{attribute 'qualified_only'}
VAR_GLOBAL
	fbManualController : FB_ManualController;
END_VAR

(* stored: Version 1.1.0.1, ProductVersion 3.1.4024.11
   GVL GVL_Devices: Id {f2d1b194-01a6-0e4d-04d9-21646c078137} *)
